// SIMATIC S7-200 SMART project (STEP 7-Micro/WIN SMART), CPU ST40

SYMBOL_TABLE System Symbols
Always_On        SM0.0    // Always ON
END_SYMBOL_TABLE

SYMBOL_TABLE Color Fixing Symbols
OpenDoor_V       Q0.0     // Open Door Valve
CloseDoor_V      Q0.1     // Close Door Valve
Heating_VI       Q0.2     // Heating Valve In
Heating_VO       Q0.3     // Heating Valve Out
Steam_VI         Q0.4     // Steam Valve In
Steam_VO         Q0.5     // Steam Valve Out
StartingLight    Q1.0
FinishLight      Q1.1
AlarmLight       Q1.2
TimeLeft         ?0_40_0
DoorClosed_S     M10.0    // Door Closed Sensor
Temp_S           VD0      // Tempreture Sensor
Pressure_S       VD4      // Pressure Sensor
Manually_S       M0.0     // Auto / Manually Switch
Start_B          M0.1     // Start Automatical Process Button
CloseDoor_B      M0.2     // Close Door Button
StartHeating_B   M0.3     // Start Heating Process Button
CoolTheRoom_B    M0.4
OpenDoor_B       M0.5     // Open Door Button
EmergencyS_B     M0.6     // Emergency Stop Button
EmergencyR_B     M0.7     // Emergency Reset Button
_MANU            M1.0
_CD              M1.2
_HeatPID         M1.3
_Cooling         M1.4
_OD              M1.5
_EmergencyS      M1.6
_EmergencyR      M1.7
Closing          M2.0     // Closing the door
Heating          M2.1     // Heating the room
Colling          M2.2     // Colling the room
Opening          M2.3     // Opening the door
Manually_Mod     M3.0
END_SYMBOL_TABLE

ORGANIZATION_BLOCK MAIN:OB1
TITLE=PROGRAM COMMENTS
BEGIN
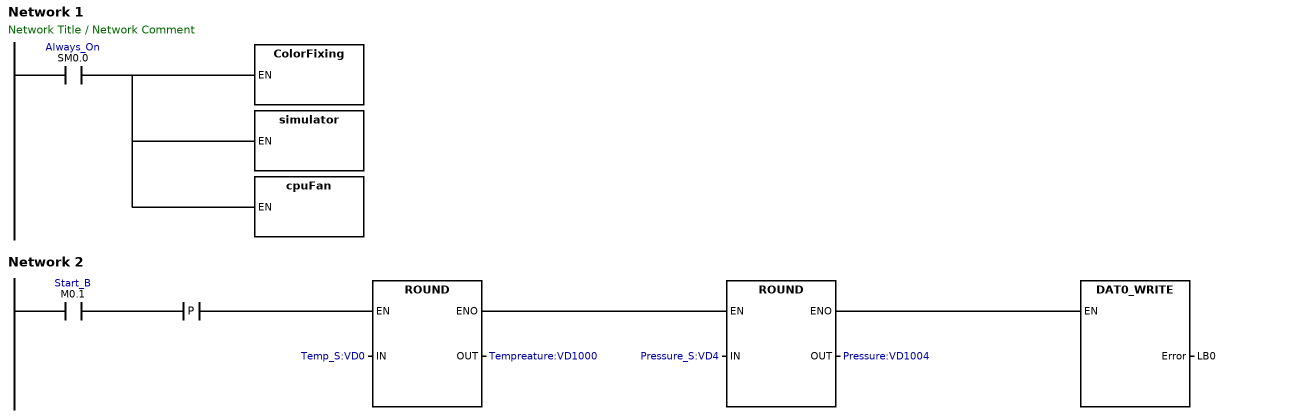
Network 1
// Network Title
// Network Comment
LD     Always_On:SM0.0
CALL   ColorFixing:SBR0
CALL   simulator:SBR10
CALL   cpuFan:SBR20
Network 2
LD     Start_B:M0.1
EU
ROUND  Temp_S:VD0, Tempreature:VD1000
AENO
ROUND  Pressure_S:VD4, Pressure:VD1004
AENO
CALL   DAT0_WRITE:SBR1, LB0
END_ORGANIZATION_BLOCK

SUBROUTINE_BLOCK ColorFixing:SBR0
TITLE=SUBROUTINE COMMENTS
BEGIN
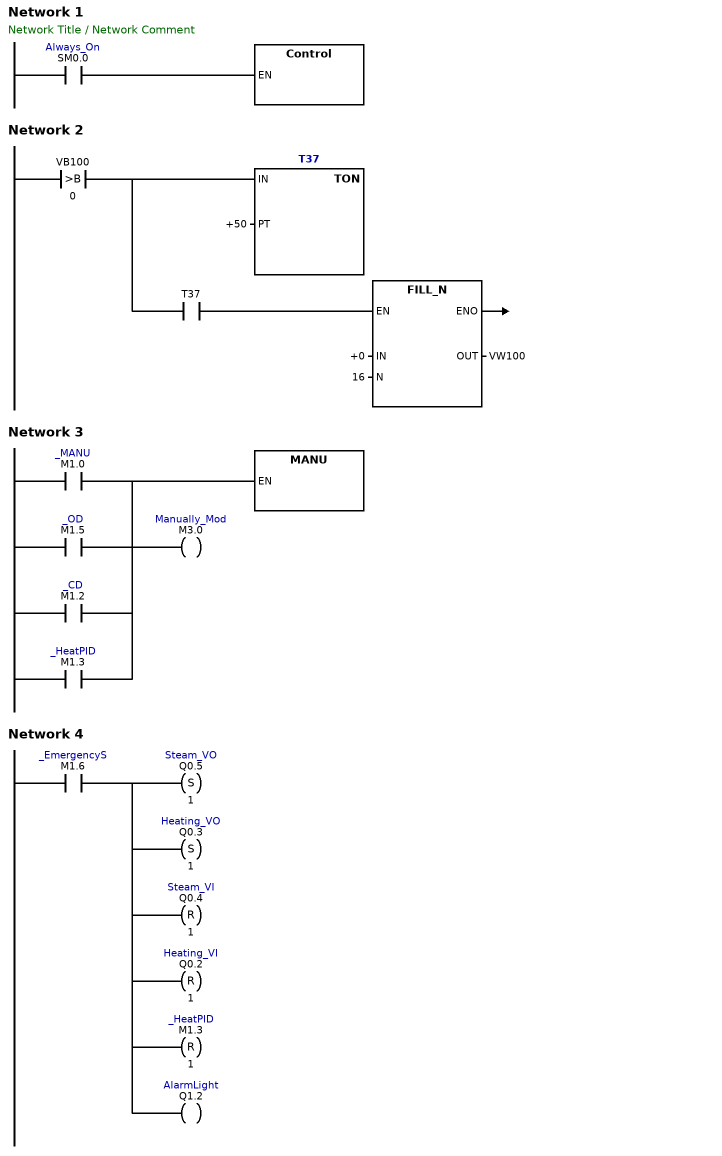
Network 1
// Network Title
// Network Comment
LD     Always_On:SM0.0
CALL   Control:SBR9
Network 2
LDB>   VB100, 0
TON    T37, +50
A      T37
FILL   +0, VW100, 16
Network 3
LD     _MANU:M1.0
O      _OD:M1.5
O      _CD:M1.2
O      _HeatPID:M1.3
CALL   MANU:SBR2
=      Manually_Mod:M3.0
Network 4
LD     _EmergencyS:M1.6
S      Steam_VO:Q0.5, 1
S      Heating_VO:Q0.3, 1
R      Steam_VI:Q0.4, 1
R      Heating_VI:Q0.2, 1
R      _HeatPID:M1.3, 1
=      AlarmLight:Q1.2
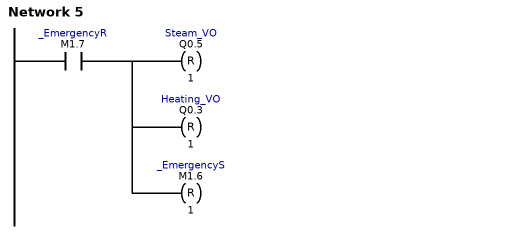
Network 5
LD     _EmergencyR:M1.7
R      Steam_VO:Q0.5, 1
R      Heating_VO:Q0.3, 1
R      _EmergencyS:M1.6, 1
END_SUBROUTINE_BLOCK

// SBR1: protected block, not included

SUBROUTINE_BLOCK MANU:SBR2
TITLE=
BEGIN
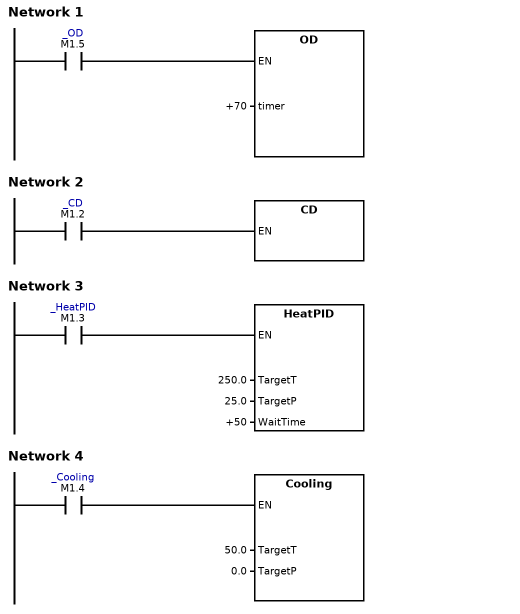
Network 1
LD     _OD:M1.5
CALL   OD:SBR3, +70
Network 2
LD     _CD:M1.2
CALL   CD:SBR4
Network 3
LD     _HeatPID:M1.3
CALL   HeatPID:SBR5, 250.0, 25.0, +50
Network 4
LD     _Cooling:M1.4
CALL   Cooling:SBR6, 50.0, 0.0
END_SUBROUTINE_BLOCK

SUBROUTINE_BLOCK OD:SBR3
TITLE=
VAR_INPUT
timer:INT;	// LW0 
END_VAR
BEGIN
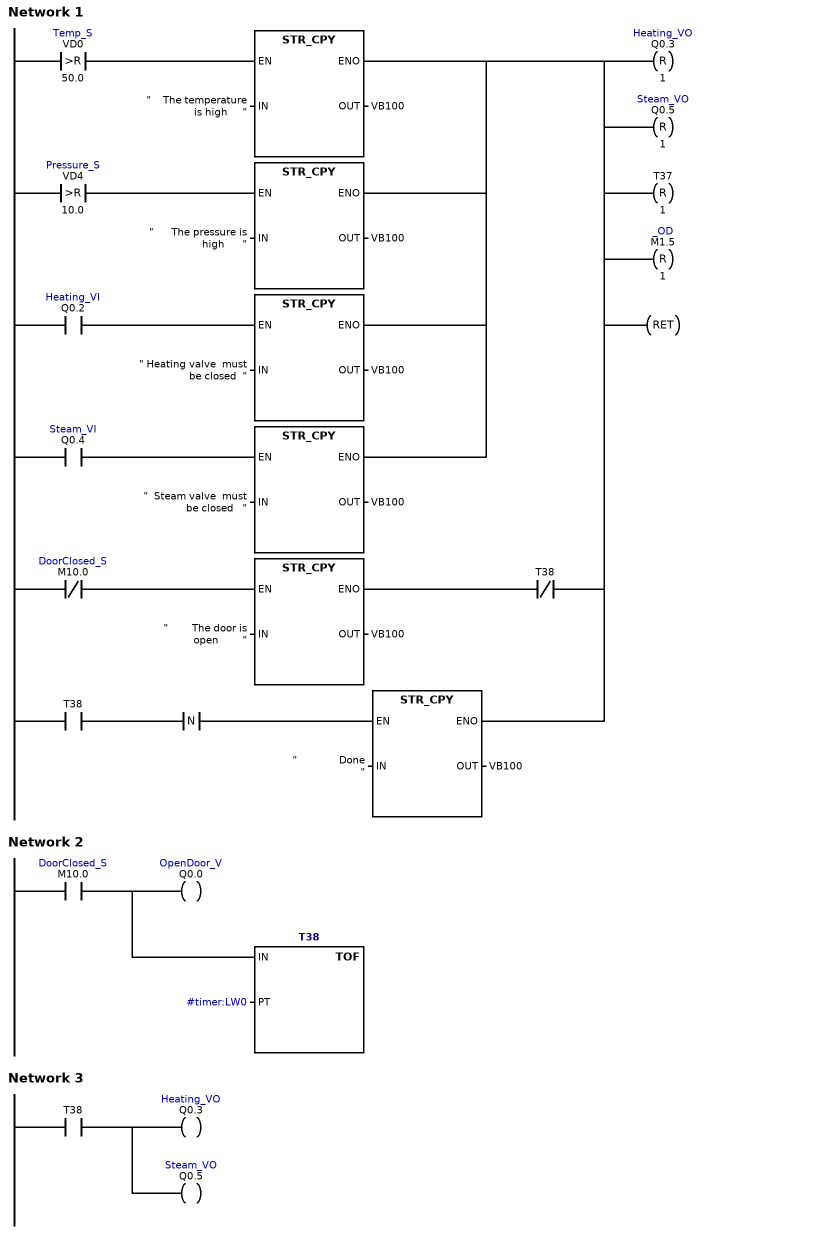
Network 1
LDR>   Temp_S:VD0, 50.0
SCPY   "    The temperature is high     ", VB100
AENO
LDR>   Pressure_S:VD4, 10.0
SCPY   "      The pressure is high      ", VB100
AENO
OLD
LD     Heating_VI:Q0.2
SCPY   " Heating valve  must be closed  ", VB100
AENO
OLD
LD     Steam_VI:Q0.4
SCPY   "  Steam valve  must be closed   ", VB100
AENO
OLD
LDN    DoorClosed_S:M10.0
SCPY   "        The door is open        ", VB100
AENO
AN     T38
OLD
LD     T38
ED
SCPY   "              Done              ", VB100
AENO
OLD
R      Heating_VO:Q0.3, 1
R      Steam_VO:Q0.5, 1
R      T37, 1
R      _OD:M1.5, 1
CRET
Network 2
LD     DoorClosed_S:M10.0
=      OpenDoor_V:Q0.0
TOF    T38, #timer:LW0
Network 3
LD     T38
=      Heating_VO:Q0.3
=      Steam_VO:Q0.5
END_SUBROUTINE_BLOCK

SUBROUTINE_BLOCK CD:SBR4
TITLE=
BEGIN
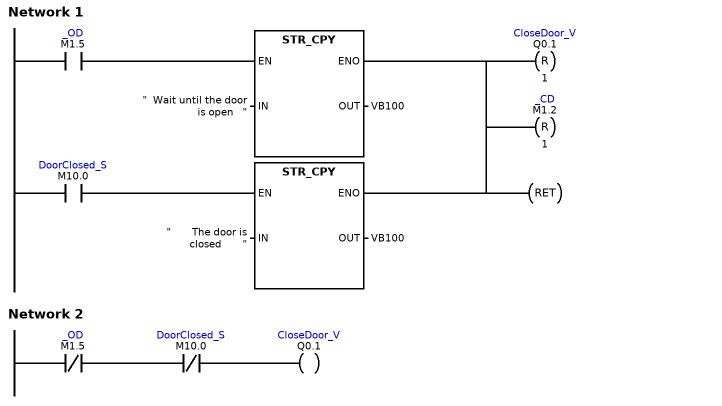
Network 1
LD     _OD:M1.5
SCPY   "  Wait until the door is open   ", VB100
AENO
LD     DoorClosed_S:M10.0
SCPY   "       The door is closed       ", VB100
AENO
OLD
R      CloseDoor_V:Q0.1, 1
R      _CD:M1.2, 1
CRET
Network 2
LDN    _OD:M1.5
AN     DoorClosed_S:M10.0
=      CloseDoor_V:Q0.1
END_SUBROUTINE_BLOCK

SUBROUTINE_BLOCK HeatPID:SBR5
TITLE=
VAR_INPUT
TargetT:REAL;	// LD0 
TargetP:REAL;	// LD4 
WaitTime:INT;	// LW8 
END_VAR
BEGIN
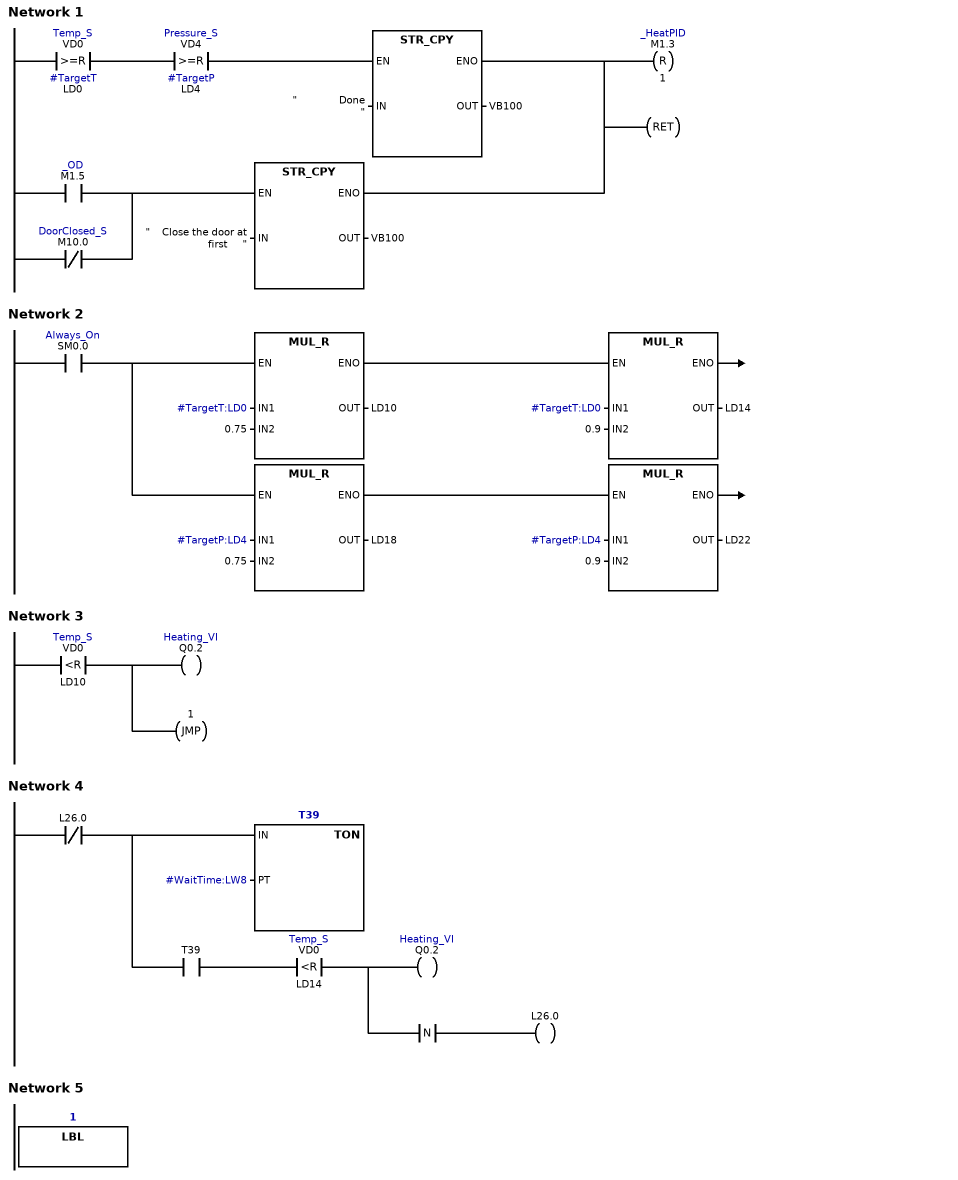
Network 1
LDR>=  Temp_S:VD0, #TargetT:LD0
AR>=   Pressure_S:VD4, #TargetP:LD4
SCPY   "              Done              ", VB100
AENO
LD     _OD:M1.5
ON     DoorClosed_S:M10.0
SCPY   "    Close the door at first     ", VB100
AENO
OLD
R      _HeatPID:M1.3, 1
CRET
Network 2
LD     Always_On:SM0.0
LPS
MOVR   #TargetT:LD0, LD10
AENO
*R     0.75, LD10
AENO
MOVR   #TargetT:LD0, LD14
*R     0.9, LD14
LPP
MOVR   #TargetP:LD4, LD18
AENO
*R     0.75, LD18
AENO
MOVR   #TargetP:LD4, LD22
*R     0.9, LD22
Network 3
LDR<   Temp_S:VD0, LD10
=      Heating_VI:Q0.2
JMP    1
Network 4
LDN    L26.0
TON    T39, #WaitTime:LW8
A      T39
AR<    Temp_S:VD0, LD14
=      Heating_VI:Q0.2
ED
=      L26.0
Network 5
LBL    1
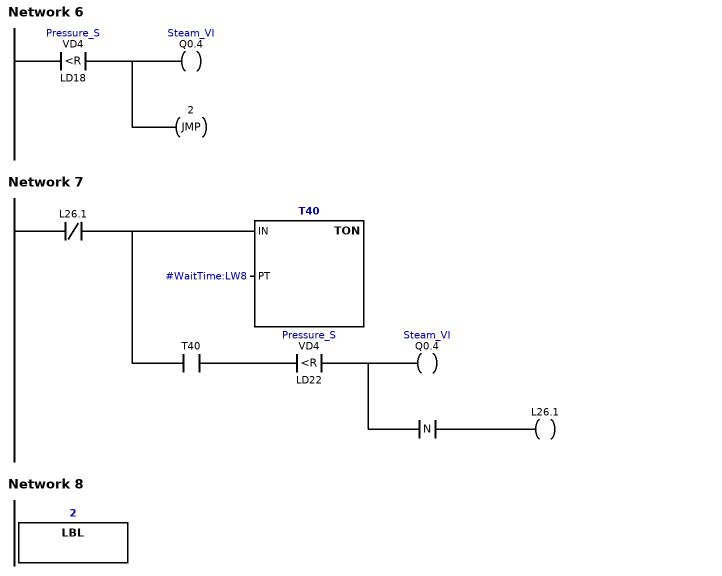
Network 6
LDR<   Pressure_S:VD4, LD18
=      Steam_VI:Q0.4
JMP    2
Network 7
LDN    L26.1
TON    T40, #WaitTime:LW8
A      T40
AR<    Pressure_S:VD4, LD22
=      Steam_VI:Q0.4
ED
=      L26.1
Network 8
LBL    2
END_SUBROUTINE_BLOCK

SUBROUTINE_BLOCK Cooling:SBR6
TITLE=
VAR_INPUT
TargetT:REAL;	// LD0 
TargetP:REAL;	// LD4 
END_VAR
BEGIN
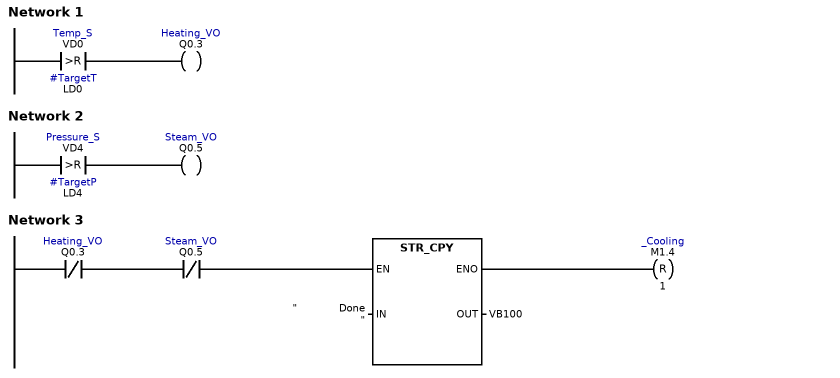
Network 1
LDR>   Temp_S:VD0, #TargetT:LD0
=      Heating_VO:Q0.3
Network 2
LDR>   Pressure_S:VD4, #TargetP:LD4
=      Steam_VO:Q0.5
Network 3
LDN    Heating_VO:Q0.3
AN     Steam_VO:Q0.5
SCPY   "              Done              ", VB100
AENO
R      _Cooling:M1.4, 1
END_SUBROUTINE_BLOCK

// SBR7: protected block, not included

SUBROUTINE_BLOCK Control:SBR9
TITLE=
BEGIN
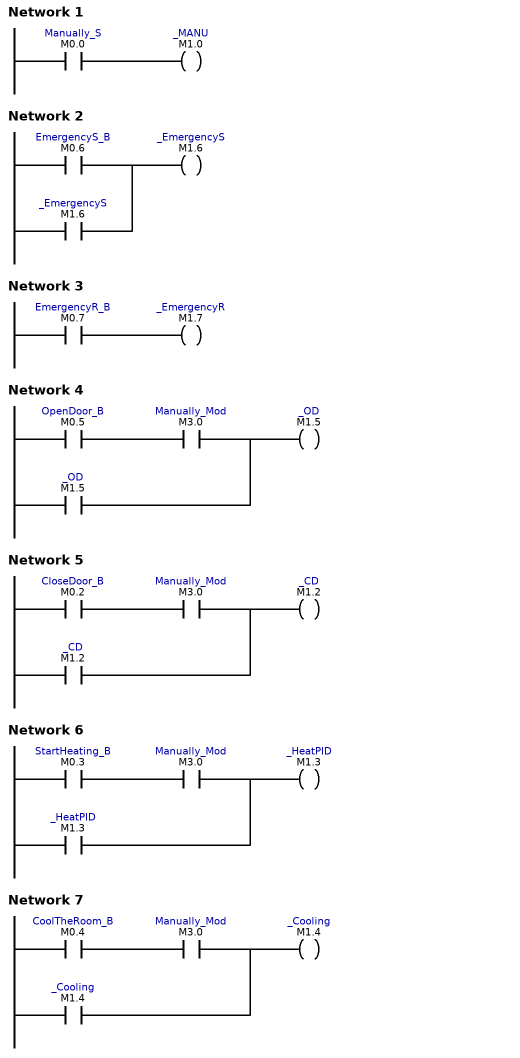
Network 1
LD     Manually_S:M0.0
=      _MANU:M1.0
Network 2
LD     EmergencyS_B:M0.6
O      _EmergencyS:M1.6
=      _EmergencyS:M1.6
Network 3
LD     EmergencyR_B:M0.7
=      _EmergencyR:M1.7
Network 4
LD     OpenDoor_B:M0.5
A      Manually_Mod:M3.0
O      _OD:M1.5
=      _OD:M1.5
Network 5
LD     CloseDoor_B:M0.2
A      Manually_Mod:M3.0
O      _CD:M1.2
=      _CD:M1.2
Network 6
LD     StartHeating_B:M0.3
A      Manually_Mod:M3.0
O      _HeatPID:M1.3
=      _HeatPID:M1.3
Network 7
LD     CoolTheRoom_B:M0.4
A      Manually_Mod:M3.0
O      _Cooling:M1.4
=      _Cooling:M1.4
END_SUBROUTINE_BLOCK

SUBROUTINE_BLOCK simulator:SBR10
TITLE=
BEGIN
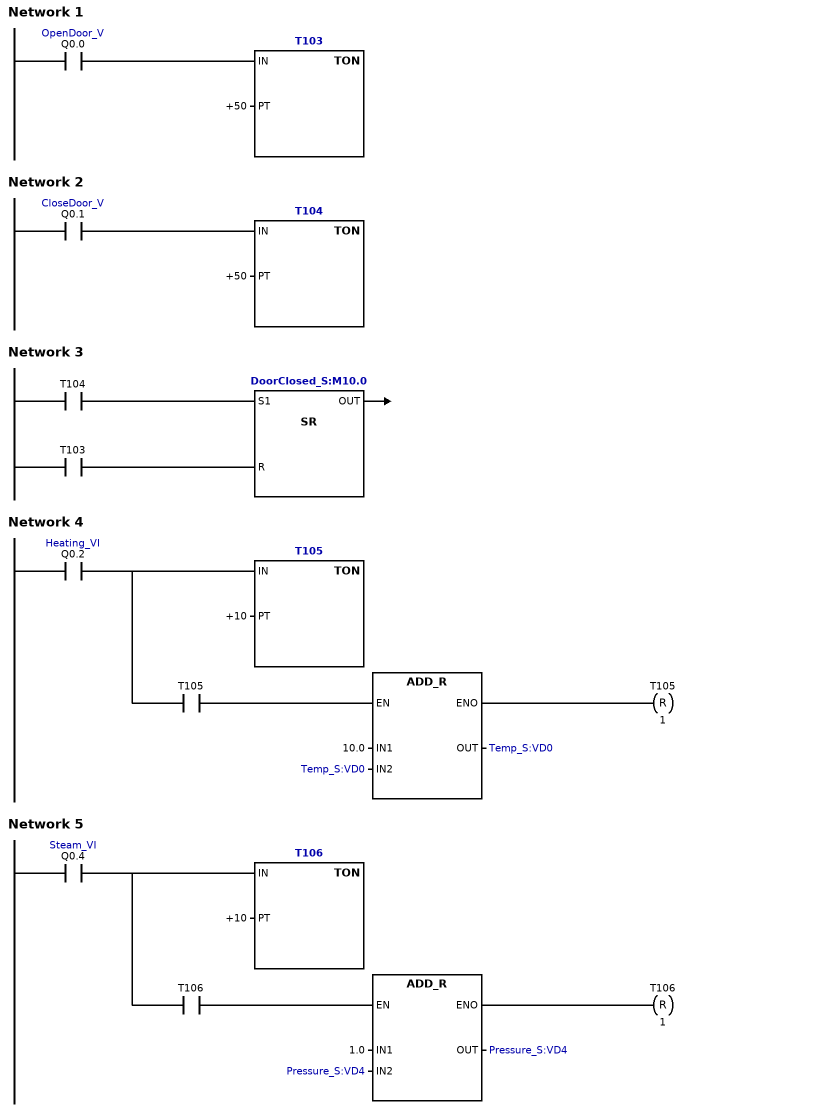
Network 1
LD     OpenDoor_V:Q0.0
TON    T103, +50
Network 2
LD     CloseDoor_V:Q0.1
TON    T104, +50
Network 3
LD     T104
LD     T103
NOT
A      DoorClosed_S:M10.0
OLD
=      DoorClosed_S:M10.0
Network 4
LD     Heating_VI:Q0.2
TON    T105, +10
A      T105
+R     10.0, Temp_S:VD0
AENO
R      T105, 1
Network 5
LD     Steam_VI:Q0.4
TON    T106, +10
A      T106
+R     1.0, Pressure_S:VD4
AENO
R      T106, 1
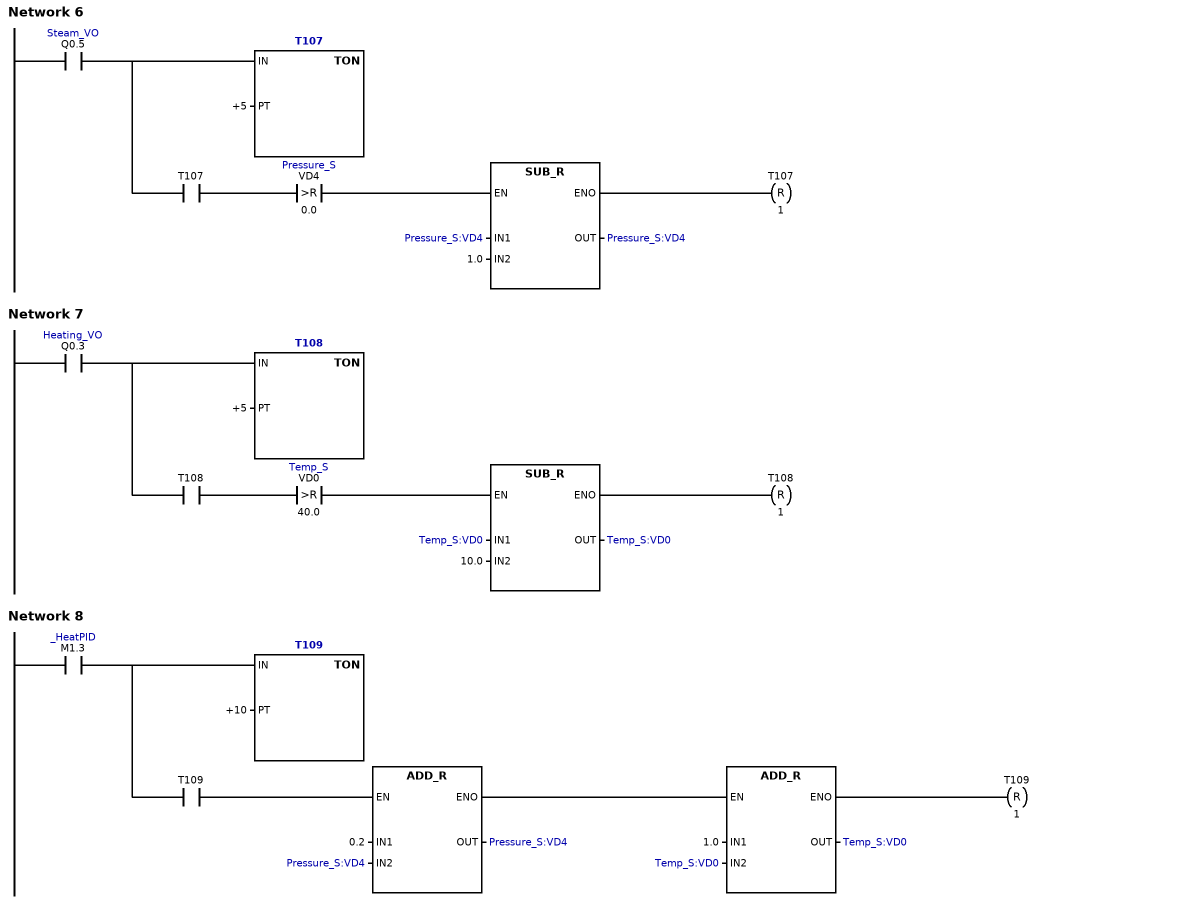
Network 6
LD     Steam_VO:Q0.5
TON    T107, +5
A      T107
AR>    Pressure_S:VD4, 0.0
-R     1.0, Pressure_S:VD4
AENO
R      T107, 1
Network 7
LD     Heating_VO:Q0.3
TON    T108, +5
A      T108
AR>    Temp_S:VD0, 40.0
-R     10.0, Temp_S:VD0
AENO
R      T108, 1
Network 8
LD     _HeatPID:M1.3
TON    T109, +10
A      T109
+R     0.2, Pressure_S:VD4
AENO
+R     1.0, Temp_S:VD0
AENO
R      T109, 1
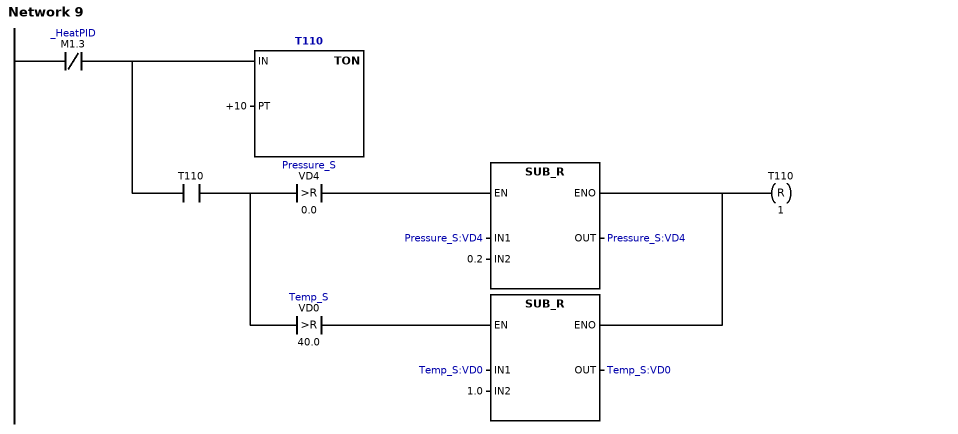
Network 9
LDN    _HeatPID:M1.3
TON    T110, +10
A      T110
LPS
AR>    Pressure_S:VD4, 0.0
-R     0.2, Pressure_S:VD4
AENO
=      L63.7
LPP
AR>    Temp_S:VD0, 40.0
-R     1.0, Temp_S:VD0
AENO
O      L63.7
R      T110, 1
END_SUBROUTINE_BLOCK

SUBROUTINE_BLOCK cpuFan:SBR20
TITLE=
BEGIN
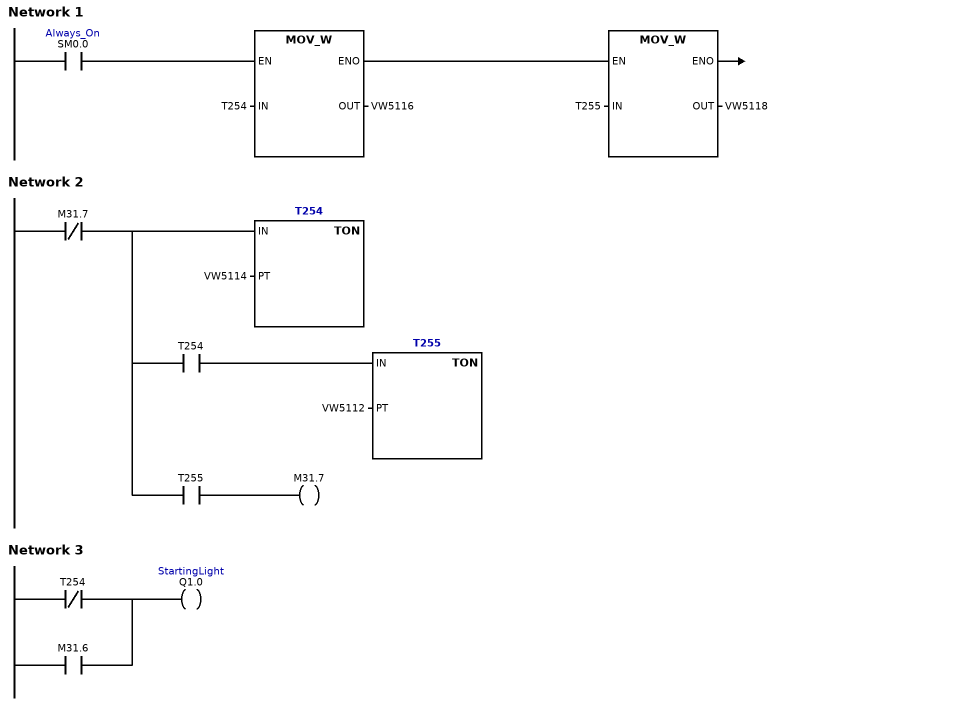
Network 1
LD     Always_On:SM0.0
MOVW   T254, VW5116
AENO
MOVW   T255, VW5118
Network 2
LDN    M31.7
LPS
TON    T254, VW5114
A      T254
TON    T255, VW5112
LPP
A      T255
=      M31.7
Network 3
LDN    T254
O      M31.6
=      StartingLight:Q1.0
END_SUBROUTINE_BLOCK
